FUNCTION CheckCalculation : LREAL
VAR_INPUT
  otg : Struckig.IOtg;
END_VAR

REPEAT 
  otg.Cyclic();
  otg.PassOutputToInput();
UNTIL otg.State <> Struckig.TrajectoryState.Busy END_REPEAT

CheckCalculation := otg.Duration;

END_FUNCTION

(* stored: Version 1.1.0.1
   POU CheckCalculation: Id {7705c60f-b3f4-4b53-bef5-2ced749a7c74}, SpecialFunc None *)
